// TIA Portal V21 export
VAR_GLOBAL   // PLC tag table "K_Tipo"
END_VAR
VAR_GLOBAL CONSTANT   // user constants
   K_TipoAnalogica : Int := 1;
   K_TipoPid : Int := 2;
   K_TipoPortata : Int := 3;
   K_TipoTrend : Int := 4;
   K_TipoParatia : Int := 5;
   K_TipoMotore : Int := 6;
   K_TipoAllarme : Int := 7;
   K_TipoValvola : Int := 8;
   K_TipoSezionePastorizzatore : Int := 9;
   K_TipoZona : Int := 10;
   K_TipoComunicazione : Int := 11;
   K_TipoSequenza : Int := 12;
   K_TipoSegnaliMacchine : Int := 13;
   K_TipoSensore : Int := 14;
   K_TipoAdditivo : Int := 15;
   K_TipoRicetta : Int := 16;
   K_TipoStazione : Int := 17;
END_VAR
